FUNCTION_BLOCK FB_ModbusTCPIP_ReadCoils

VAR

fbMBReadCoils : FB_MBReadCoils ;
nReadValue : BYTE;

eReadState : (WAIT, TRIGGER,READ);
fbTrigger : R_TRIG;
END_VAR

fbTrigger();
IF fbTrigger.Q THEN
	IF eReadState = WAIT THEN 
	eReadState := TRIGGER;
	END_IF
END_IF


CASE eReadState OF
	
	WAIT :
	
	// Do nothing
	
	
	TRIGGER :
	
		fbMBReadCoils(
		
		sIPAddr   := '192.168.1.175',
		nTCPPort  := 502,
		nUnitID   := 16#FF,
		nQuantity := 1,
		nMBAddr   := 0,
		cbLength  := SIZEOF(nReadValue),
		pDestAddr := ADR(nReadValue),
		bExecute  := TRUE,
		tTimeout  :=T#5S,
		bBusy=>,
		bError=>,
		nErrId=>,
		cbRead=>,
						);
		eReadState := READ;
	
	READ :
	
	// Here we will be waiting for the response
		fbMBReadCoils(bExecute := FALSE);
		IF NOT fbMBReadCoils.bBusy OR fbMBReadCoils.bError THEN
			eReadState :=WAIT;
			
		END_IF
		
END_CASE

END_FUNCTION_BLOCK

(* stored: Version 1.1.0.1, ProductVersion 3.1.4024.11
   POU FB_ModbusTCPIP_ReadCoils: Id {6eabe492-3d96-4fc3-85ca-686ce9fb6388}, SpecialFunc None *)
